PROGRAM PRG_Task3
VAR
	{attribute 'displaymode':='hex'} 
	CallingTaskAdsPort :UINT;	
END_VAR

CallingTaskAdsPort:=_TaskInfo[GETCURTASKINDEXEX()].AdsPort;

IF GVL.fbCrititcalSection.Enter() THEN
	(* start of critical section *)
	GVL.fbDoWork.M_ConsumeTime(CallerTaskAdsPort :=CallingTaskAdsPort );

	(* end of critical section *)
	GVL.fbCrititcalSection.Leave();
END_IF

END_PROGRAM

(* stored: Version 1.1.0.1, ProductVersion 3.1.4026.18
   POU PRG_Task3: Id {f6513162-bf51-4efc-9900-3629ed9bc665}, SpecialFunc None *)
